% RSLogix 500 project PROJECT 1  CGT part 2.RSS, saved by version 8.30.00.16 %
PROJECT "UNTITLED"    % processor: Bul.1763 MicroLogix 1100 Series B %

PROGRAM FILES
  LAD 2 "MAIN"  4 rungs
  LAD 3 "INPUTS"  3 rungs
  LAD 4 "LOGIC"  10 rungs
  LAD 5 "OUTPUTS"  3 rungs

DATA FILES
  O0 OUTPUT  4 elements
  I1 INPUT  6 elements
  S2 STATUS  66 elements
  B3 BINARY  1 elements
  T4 TIMER  1 elements
  C5 COUNTER  1 elements
  R6 CONTROL  1 elements
  N7 INTEGER  1 elements
  F8 FLOAT  1 elements

LADDER 2 "MAIN"
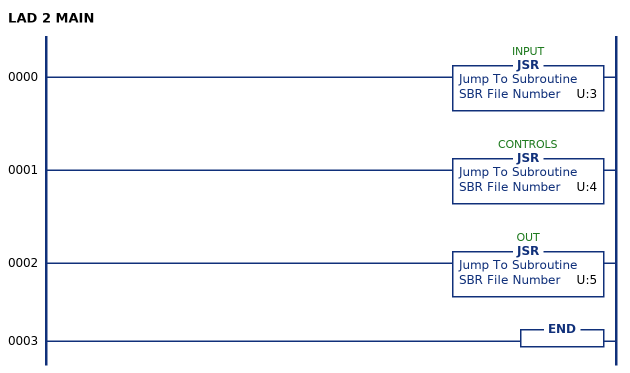
% Rung: 0 %  % edit flag set %
SOR JSR U:3 EOR
%   U:3  "INPUT" %
% Rung: 1 %  % edit flag set %
SOR JSR U:4 EOR
%   U:4  "CONTROLS" %
% Rung: 2 %  % edit flag set %
SOR JSR U:5 EOR
%   U:5  "OUT" %
% Rung: 3 %
SOR END EOR

LADDER 3 "INPUTS"
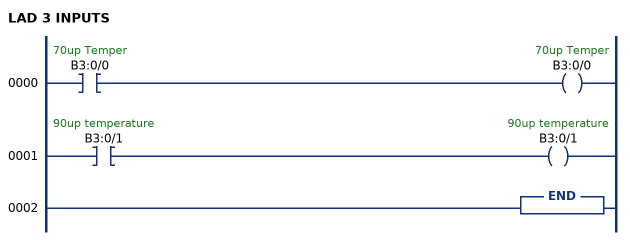
% Rung: 0 %  % edit flag set %
SOR XIC B3:0/0 OTE B3:0/0 EOR
%   B3:0/0  "70up Temper" %
% Rung: 1 %  % edit flag set %
SOR XIC B3:0/1 OTE B3:0/1 EOR
%   B3:0/1  "90up temperature" %
% Rung: 2 %
SOR END EOR

LADDER 4 "LOGIC"
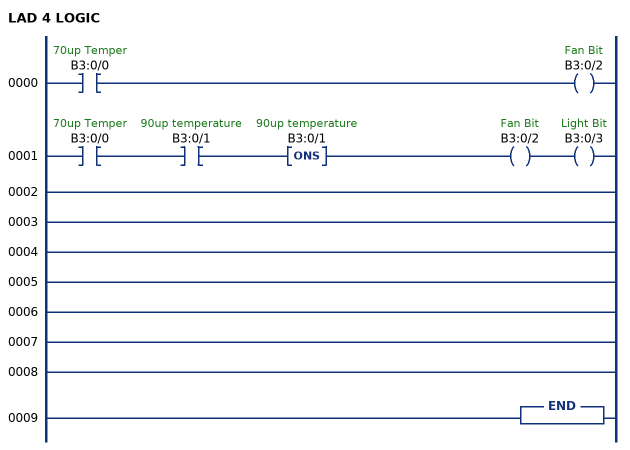
% Rung: 0 %  % edit flag set %
SOR XIC B3:0/0 OTE B3:0/2 EOR
%   B3:0/0  "70up Temper" %
%   B3:0/2  "Fan Bit" %
% Rung: 1 %  % edit flag set %
SOR XIC B3:0/0 XIC B3:0/1 ONS B3:0/1 OTE B3:0/2 OTE B3:0/3 EOR
%   B3:0/0  "70up Temper" %
%   B3:0/1  "90up temperature" %
%   B3:0/2  "Fan Bit" %
%   B3:0/3  "Light Bit" %
% Rung: 2 %  % edit flag set %
SOR EOR
% Rung: 3 %  % edit flag set %
SOR EOR
% Rung: 4 %  % edit flag set %
SOR EOR
% Rung: 5 %  % edit flag set %
SOR EOR
% Rung: 6 %  % edit flag set %
SOR EOR
% Rung: 7 %  % edit flag set %
SOR EOR
% Rung: 8 %  % edit flag set %
SOR EOR
% Rung: 9 %
SOR END EOR

LADDER 5 "OUTPUTS"
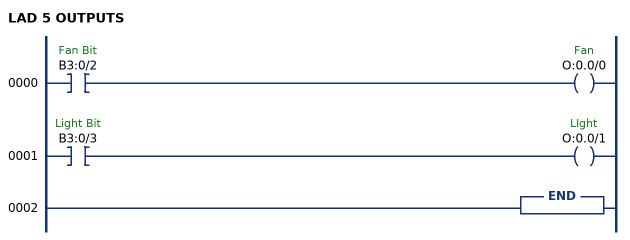
% Rung: 0 %
SOR XIC B3:0/2 OTE O:0.0/0 EOR
%   B3:0/2  "Fan Bit" %
%   O:0.0/0  "Fan" %
% Rung: 1 %
SOR XIC B3:0/3 OTE O:0.0/1 EOR
%   B3:0/3  "Light Bit" %
%   O:0.0/1  "LIght" %
% Rung: 2 %
SOR END EOR
